{attribute addProperty BoxType "APS4322-7000-0017"}
{attribute addProperty Id "CommStatusWordAT %I*UINT16217DataAT %I*ARRAY[0 ..3] OF UINT6480"}
{attribute addProperty CRC "3217752388"}
{attribute addProperty SizeInBites "80"}
{attribute addProperty SizeInBytes "10"}
TYPE APS_Comm_Inputs_FF1CE56E :
STRUCT
	{attribute addProperty Name "CommStatusWord"}
	CommStatusWord AT %I* : UINT;
	{attribute addProperty Name "Data"}
	Data AT %I* : ARRAY[0 ..3] OF UINT;
END_STRUCT
END_TYPE

(* stored: Version 1.2.0.0, ProductVersion 3.1.4024.9
   DUT APS_Comm_Inputs_FF1CE56E: Id {7574ac90-ddd6-4572-a34d-32fd2031e05e} *)
